FUNCTION_BLOCK PUBLIC clsStringBuilder IMPLEMENTS  I_StringBuilder, I_LimitedStringBuilder
VAR
	{attribute 'hide'}
	_workString : STRING;
END_VAR

METHOD PUBLIC Append : I_StringBuilder // Append text to t current build string.
VAR_INPUT
	Text : STRING; //Text to append to current build string
END_VAR
_workString:= CONCAT(_WorkString, Text);
Append := THIS^;
END_METHOD

METHOD PUBLIC InsertAtLocation : I_StringBuilder
VAR_INPUT
	Text : STRING;
	Position : INT;
END_VAR
_WorkString := Tc2_Standard.INSERT(_WorkSTring, Text, Position);
InsertAtLocation := THIS^;
END_METHOD

METHOD PUBLIC Left : I_StringBuilder
VAR_INPUT
	Count	: INT;
END_VAR
_workString:= Tc2_Standard.LEFT(_WorkString, Count);
Left := THIS^;
END_METHOD

PROPERTY Length : INT
GET
Length := LEN(_workString);
END_GET
END_PROPERTY

METHOD PUBLIC Reset : I_LimitedStringBuilder // Reset current build string to an empty string.
_WorkString := '';
Reset := THIS^;
END_METHOD

METHOD Right : I_StringBuilder
VAR_INPUT
	Count	: INT;
END_VAR
_workString:= Tc2_Standard.RIGHT(_WorkString, Count);
Right := THIS^;
END_METHOD

METHOD PUBLIC ToString : STRING //Returns current build string.
ToString := _WorkString;
END_METHOD

END_FUNCTION_BLOCK

(* stored: Version 1.1.0.1, ProductVersion 3.1.4024.12
   POU clsStringBuilder: Id {368e5049-935b-4562-a874-cb9be5225f7d}, SpecialFunc None
   Method Append: Id {3f45997e-6006-457f-9a9a-30ac281e8f8a}
   Method InsertAtLocation: Id {b2ed9ced-aca1-4991-af8e-c808997da606}
   Method Left: Id {eedcf736-2954-4be2-9a10-4eef313e2edc}
   Property Length: Id {1625b249-2c40-493a-91b2-4f976cbd13c7}
   Get Get: Id {69f820ae-44d5-4ad7-94ba-447bf8f9e353}
   Method Reset: Id {f04f2676-7659-44a8-87c7-48fdd5328c04}
   Method Right: Id {378f0fdc-3469-4c64-8653-911bf890f042}
   Method ToString: Id {8c20dc6d-f3fa-4203-b887-d1b9b96ecacc} *)
